FUNCTION_BLOCK FB_CH_List EXTENDS FB_CH_Object IMPLEMENTS I_CH_LIST, I_CH_List_Dublicate
VAR
	{attribute 'hide'}
	nObjectCount			: UDINT;
	{attribute 'hide'}
	nIdxNextObject			: UDINT;
	{attribute 'hide'}
	nIdxLastRestoreValues : ARRAY [0..(MAX_CTS_RESTORE_VALUES+1)] OF UDINT;
	{attribute 'hide'}
	nIdxRestore				: UDINT;
	{attribute 'hide'}
	aObjects				: ARRAY [1..BaseParameterlist.MAX_OBJECTS] OF I_CH_Object;
END_VAR
VAR CONSTANT
	{attribute 'hide'}
	MAX_CTS_RESTORE_VALUES : UINT := 20;
END_VAR

//Add all objects from the list in to this list
METHOD PUBLIC AddList : HRESULT
VAR_INPUT
	ipList	: I_CH_List;
END_VAR
VAR
	hr : HRESULT;
	ipListDublicate : I_CH_List_Dublicate;
	refRemoteList : REFERENCE TO ARRAY [1..BaseParameterlist.MAX_OBJECTS] OF I_CH_Object;
	pRemoteList : PVOID;
END_VAR
VAR_INST
	{attribute 'hide'}
	fbAlarmInvalideInputparm : FB_TcAlarm;
	{attribute 'hide'}
	fbAlarmListToSmall : FB_TcAlarm;
END_VAR
// Invalide input
IF ipList = 0 THEN
	fbAlarmInvalideInputparm.CreateEx(stEventEntry:= TC_EVENTS.CHALET_Base_Events.Invalide_Inputparameter, 
							ipSourceInfo := THIS^.fbSourceInfo, 
							bWithConfirmation := FALSE);
	fbAlarmInvalideInputparm.ipArguments.Clear().AddStringByValue('ipList');
	fbAlarmInvalideInputparm.Raise(0);	

	AddList := S_FALSE;
	RETURN;
END_IF


// This list is to small
IF (ipList.Size + THIS^.Size) > BaseParameterlist.MAX_OBJECTS THEN
	fbAlarmListToSmall.CreateEx(stEventEntry:= TC_EVENTS.CHALET_Base_Events.ListIsToSmall, 
							ipSourceInfo := THIS^.fbSourceInfo, 
							bWithConfirmation := FALSE);
	fbAlarmListToSmall.Raise(0);	

	AddList := S_FALSE;
	RETURN;
END_IF


//Done nothing to add
IF ipList.Size = 0 THEN
	AddList := S_OK;
	RETURN;
END_IF


//Check if the list has an optional I_CH_List_Dublicate interface. If so use the faste memcpy, else use default list commands
IF __QUERYINTERFACE(ipList, ipListDublicate) AND_THEN __ISVALIDREF(ipListDublicate.Content) THEN
	refRemoteList REF= ipListDublicate.Content;
	pRemoteList := ADR(refRemoteList);
	Tc2_System.MEMCPY(destAddr:= ADR(THIS^.aObjects[(THIS^.nObjectCount+1)]), srcAddr:= pRemoteList, n:= (SIZEOF(THIS^.aObjects[1])*ipList.Size) );
	THIS^.nObjectCount := ipList.Size + THIS^.nObjectCount; //Set size of List
ELSE
	ipList.ResetIterator();
	WHILE ipList.HasNextObject() DO
		hr := THIS^.AddObject(ipList.GetNextObject());
		IF hr <> S_OK THEN
			//Error
			AddList := hr;
			RETURN;
		END_IF
	END_WHILE
	ipList.RestoreIterator();
END_IF
END_METHOD

METHOD PUBLIC AddObject : HRESULT
VAR_INPUT
	iChObject	: I_CH_Object;
END_VAR
VAR_INST
	{attribute 'hide'}
	fbAlarmListFull : FB_TcAlarm;
END_VAR
IF iChObject = 0 THEN
	AddObject := S_FALSE;
	RETURN;
END_IF


//Error if list is allready full
IF nObjectCount >= BaseParameterlist.MAX_OBJECTS THEN
	fbAlarmListFull.CreateEx(stEventEntry:= TC_EVENTS.CHALET_Base_Events.ListIsFull, 
							ipSourceInfo := THIS^.fbSourceInfo, 
							bWithConfirmation := FALSE);
	fbAlarmListFull.ipArguments.Clear().AddStringByValue(iChObject.LUID);
	fbAlarmListFull.Raise(0);
	AddObject := S_FALSE;
	RETURN;
END_IF


//Add to list
nObjectCount := nObjectCount + 1;
aObjects[nObjectCount] := iChObject;

AddObject := S_OK;
END_METHOD

METHOD PUBLIC Clear : BOOL
VAR
	nIdx : UDINT;
END_VAR
Tc2_System.MEMSET(	destAddr	:= ADR(aObjects[1]), 
					fillByte	:= 0, 
					n			:= SIZEOF(aObjects[1])*BaseParameterlist.MAX_OBJECTS);


nObjectCount	:= 0;
nIdxNextObject	:= 0;
END_METHOD

//DEBUG only. View content for easy debug. Do not use this property
{attribute 'monitoring':='call'}
PROPERTY Content : REFERENCE TO ARRAY [1..BaseParameterlist.MAX_OBJECTS] OF I_CH_Object
GET
Content REF= THIS^.aObjects;
END_GET
END_PROPERTY

METHOD Duplicate : BOOL
VAR_INPUT
	ipListCopyFrom : I_CH_LIST;
END_VAR
VAR
	ipThisList : I_CH_LIST := THIS^;
	hr : HRESULT;
	ipListDublicate : I_CH_List_Dublicate;
	refRemoteList : REFERENCE TO ARRAY [1..BaseParameterlist.MAX_OBJECTS] OF I_CH_Object;
	pRemoteList : PVOID;
END_VAR
VAR_INST
	{attribute 'hide'}
	fbAlarmInvalideInputparm : FB_TcAlarm;
	{attribute 'hide'}
	fbAlarmListToSmall : FB_TcAlarm;
END_VAR
//New list equals this list
IF ipListCopyFrom = ipThisList THEN
	//Do Nothing - Successfull
	Duplicate := TRUE;
	RETURN;
END_IF

THIS^.Clear();

// Invalide input
IF ipListCopyFrom = 0 THEN
	fbAlarmInvalideInputparm.CreateEx(stEventEntry:= TC_EVENTS.CHALET_Base_Events.Invalide_Inputparameter, 
							ipSourceInfo := THIS^.fbSourceInfo, 
							bWithConfirmation := FALSE);
	fbAlarmInvalideInputparm.ipArguments.Clear().AddStringByValue('ipListCopyFrom');
	fbAlarmInvalideInputparm.Raise(0);	

	Duplicate := FALSE;
	RETURN;
END_IF


// This list is to small
IF ipListCopyFrom.Size > BaseParameterlist.MAX_OBJECTS THEN
	fbAlarmListToSmall.CreateEx(stEventEntry:= TC_EVENTS.CHALET_Base_Events.ListIsToSmall, 
							ipSourceInfo := THIS^.fbSourceInfo, 
							bWithConfirmation := FALSE);
	fbAlarmListToSmall.Raise(0);	
	Duplicate := FALSE;
	RETURN;
END_IF


//Done nothing to add
IF ipListCopyFrom.Size = 0 THEN
	Duplicate := TRUE;
	RETURN;
END_IF


//Check if the list has an optional I_CH_List_Dublicate interface. If so use the faste memcpy, else use list commands
IF __QUERYINTERFACE(ipListCopyFrom, ipListDublicate) AND_THEN __ISVALIDREF(ipListDublicate.Content) THEN
	refRemoteList REF= ipListDublicate.Content;
	pRemoteList := ADR(refRemoteList);
	Tc2_System.MEMCPY(destAddr:= ADR(THIS^.aObjects), srcAddr:= pRemoteList, n:= (SIZEOF(THIS^.aObjects[1])*ipListCopyFrom.Size) );
	THIS^.nObjectCount := ipListCopyFrom.Size; //Set size of List
ELSE
	ipListCopyFrom.ResetIterator();
	WHILE ipListCopyFrom.HasNextObject() DO
		hr := THIS^.AddObject(ipListCopyFrom.GetNextObject());
		IF hr <> S_OK THEN
			//Error
			Duplicate := FALSE;
			RETURN;
		END_IF
	END_WHILE
	ipListCopyFrom.RestoreIterator();	
END_IF


Duplicate := TRUE;
END_METHOD

METHOD PUBLIC FindLUID : I_CH_OBJECT
VAR_INPUT
	sLUID	: STRING;
END_VAR
VAR
	nIdx : UDINT;
END_VAR
FOR nIdx := 1 TO nObjectCount DO
	IF aObjects[nIdx] <> 0 AND_THEN aObjects[nIdx].LUID = sLUID THEN
		FindLUID := aObjects[nIdx];
		EXIT;
	END_IF
END_FOR
END_METHOD

METHOD FindOID : I_CH_OBJECT
VAR_INPUT
	nOID	: OTCID;
END_VAR
VAR
	nIdx : UDINT;
END_VAR
FOR nIdx := 1 TO nObjectCount DO
	IF aObjects[nIdx] <> 0 AND_THEN aObjects[nIdx].OID = nOID THEN
		FindOID := aObjects[nIdx];
		EXIT;
	END_IF
END_FOR
END_METHOD

METHOD FindOIDString : I_CH_OBJECT
VAR_INPUT
	sOID	: STRING;
END_VAR
VAR
	nIdx : UDINT;
END_VAR
FOR nIdx := 1 TO nObjectCount DO
	IF aObjects[nIdx] <> 0 AND_THEN DWORD_TO_HEXSTR(TO_DWORD(aObjects[nIdx].OID),0,FALSE) = sOID THEN
		FindOIDString := aObjects[nIdx];
		EXIT;
	END_IF
END_FOR
END_METHOD

METHOD PUBLIC GetNextObject : I_CH_Object
VAR_INPUT
END_VAR
VAR_INST
	{attribute 'hide'}
	fbAlarmInvalideEndOfList : FB_TcAlarm;
END_VAR
nIdxNextObject := nIdxNextObject + 1;


IF nIdxNextObject > nObjectCount THEN
	//Error!
	fbAlarmInvalideEndOfList.CreateEx(stEventEntry:= TC_EVENTS.CHALET_Base_Events.Invalive_EndOfList, 
							ipSourceInfo := THIS^.fbSourceInfo, 
							bWithConfirmation := FALSE);
	fbAlarmInvalideEndOfList.ipArguments.Clear().AddStringByValue('.GetNextObject()');
	fbAlarmInvalideEndOfList.Raise(0);
	RETURN;
END_IF




GetNextObject := aObjects[nIdxNextObject];
END_METHOD

METHOD GetObjectWithHighestNumber : I_CH_Object

VAR
	nIdx : UDINT;
	nMaxSortNbr : UDINT;
END_VAR




//Check array until a match
FOR nIdx := 1 TO THIS^.nObjectCount DO
	IF THIS^.aObjects[nIdx].SortOrderInList >= nMaxSortNbr THEN
		GetObjectWithHighestNumber := THIS^.aObjects[nIdx];
		nMaxSortNbr := THIS^.aObjects[nIdx].SortOrderInList;
	END_IF
END_FOR
END_METHOD

METHOD GetObjectWithLowestNumber : I_CH_Object
VAR
	nIdx : UDINT;
	nMinSortNbr : UDINT := GVL_Datatypes.cMaxUDint;
END_VAR
//Check array until a match
FOR nIdx := 1 TO THIS^.nObjectCount DO
	IF THIS^.aObjects[nIdx].SortOrderInList <= nMinSortNbr THEN
		GetObjectWithLowestNumber := THIS^.aObjects[nIdx];
		nMinSortNbr := THIS^.aObjects[nIdx].SortOrderInList;
	END_IF
END_FOR
END_METHOD

METHOD GetRandomObject : I_CH_Object
VAR_INPUT
END_VAR

VAR_INST
	{attribute 'hide'}
	fbDRAN : DRAND;
END_VAR

VAR
	nRandomIdx : UDINT;
END_VAR
//Check if not Empty
IF UDINT_TO_BOOL(nObjectCount) THEN
	// Generate number 0..1
	fbDRAN(Seed:= 42);
	
	// 1..Size   = ((0..1)*(Size-1))+1
	nRandomIdx := LREAL_TO_UDINT(fbDRAN.Num * (nObjectCount-1))+1;
	
	GetRandomObject := aObjects[nRandomIdx];
	
END_IF
END_METHOD

METHOD PUBLIC HasNextObject : BOOL
VAR_INPUT
END_VAR
HasNextObject := (nIdxNextObject < nObjectCount) AND_THEN (aObjects[nIdxNextObject+1] <> 0);
END_METHOD

METHOD Initialize : HRESULT //This method calls the respective Initialize method of all contained objects
VAR_INPUT
END_VAR
VAR
	hr : HRESULT;
	nIdx : UDINT;
END_VAR
//FOR each element
FOR nIdx := 1 TO nObjectCount DO
	// DO Init
	hr := GetMostSignificant(hr, aObjects[nIdx].Initialize());
END_FOR


Initialize := hr;
END_METHOD

{attribute 'monitoring':='call'}
PROPERTY PUBLIC IsEmpty : BOOL
GET
IsEmpty := (nObjectCount = 0);
END_GET
END_PROPERTY

{attribute 'monitoring':='call'}
PROPERTY PUBLIC IsFull : BOOL
GET
IsFull := (nObjectCount = BaseParameterlist.MAX_OBJECTS);
END_GET
END_PROPERTY

METHOD PUBLIC LUIDInList : BOOL
VAR_INPUT
	sLUID	: STRING;
END_VAR
VAR
	nIdx : UDINT;
END_VAR
//Check array until a match
FOR nIdx := 1 TO THIS^.nObjectCount DO
	IF THIS^.aObjects[nIdx].LUID = sLUID THEN
		LUIDInList := TRUE;
		EXIT;
	END_IF
END_FOR
END_METHOD

METHOD PUBLIC ObjectInList : BOOL
VAR_INPUT
	iChObject	: I_CH_Object;
END_VAR
VAR
	nIdx : UDINT;
END_VAR
//Check array until a match
FOR nIdx := 1 TO THIS^.nObjectCount DO
	IF THIS^.aObjects[nIdx] = iChObject THEN
		ObjectInList := TRUE;
		EXIT;
	END_IF
END_FOR
END_METHOD

METHOD PUBLIC OIDInList : BOOL
VAR_INPUT
	nOID	: OTCID;
END_VAR
VAR
	nIdx : UDINT;
END_VAR
//Check array until a match
FOR nIdx := 1 TO THIS^.nObjectCount DO
	IF THIS^.aObjects[nIdx].OID = nOID THEN
		OIDInList := TRUE;
		EXIT;
	END_IF
END_FOR
END_METHOD

METHOD RemoveAllDuplicateObjects : HRESULT
VAR_INPUT
END_VAR
VAR
	nIdx : UDINT;
	fbTempList : FB_CH_List;
	fbFoundDublicateObjects : FB_CH_List;
END_VAR
//Check eacht element in array, if allready was added in temp list. if found, delete
FOR nIdx := 1 TO THIS^.nObjectCount DO
	
	//check if allready was found
	IF fbTempList.ObjectInList(THIS^.aObjects[nIdx]) THEN
		//Found, add to an list to delete in next step
		fbFoundDublicateObjects.AddObject(THIS^.aObjects[nIdx]);	
	ELSE
		//Not found, add to list
		fbTempList.AddObject(THIS^.aObjects[nIdx]);	
	END_IF
END_FOR


//Delete in this list
fbFoundDublicateObjects.ResetIterator();
WHILE fbFoundDublicateObjects.HasNextObject() DO
	THIS^.RemoveObject(fbFoundDublicateObjects.GetNextObject());
END_WHILE
END_METHOD

METHOD PUBLIC RemoveObject : BOOL
VAR_INPUT
	iChObject	: I_CH_Object;
END_VAR

VAR
	nIdx			: UDINT;
END_VAR
RemoveObject := FALSE;

IF iChObject = 0 THEN
	RETURN;
END_IF

IF NOT THIS^.ObjectInList(iChObject) THEN
	RETURN;
END_IF

FOR nIdx := 1 TO nObjectCount DO
	IF aObjects[nIdx] = iChObject THEN
		aObjects[nIdx] := NULL;	
		
		nObjectCount := nObjectCount - 1;
		
		// Fill up the empty slot
		MEMMOVE(ADR(aObjects[nIdx]), ADR(aObjects[nIdx + 1]), SIZEOF(aObjects[nIdx]) * (BaseParameterlist.MAX_OBJECTS - nIdx));
	
		// If pos in list is less than ListIterator, then reduce Iterator
		IF nIdx <= nIdxNextObject THEN
			nIdxNextObject := nIdxNextObject -1;
		END_IF
		
		//Finish
		RemoveObject := TRUE;
		EXIT;
			
	END_IF
END_FOR
END_METHOD

METHOD PUBLIC ResetIterator : BOOL
VAR_INPUT
END_VAR
//Store the last few index for later restore if required - Shift array +1 step
MEMMOVE(srcAddr 	:= ADR(nIdxLastRestoreValues[0]), 
		destAddr 	:= ADR(nIdxLastRestoreValues[1]), 
		n 			:= (SIZEOF(nIdxNextObject)*MAX_CTS_RESTORE_VALUES));

//Store the last few index for later restore if required - Store last value
nIdxLastRestoreValues[0] := nIdxNextObject;


nIdxNextObject := 0;
END_METHOD

//Restore the iterator to the value before the last reset. This is necessary if several while loops are placed inside each other
METHOD PUBLIC RestoreIterator : BOOL
VAR_INPUT
END_VAR
//Store the last few index for later restore if required - Restore
nIdxNextObject := nIdxLastRestoreValues[0];

//Store the last few index for later restore if required - Shift array -1 step
MEMMOVE(srcAddr 	:= ADR(nIdxLastRestoreValues[1]), 
		destAddr 	:= ADR(nIdxLastRestoreValues[0]), 
		n 			:= (SIZEOF(nIdxNextObject)*MAX_CTS_RESTORE_VALUES));
END_METHOD

{attribute 'monitoring':='call'}
PROPERTY PUBLIC Size : UDINT
GET
Size := nObjectCount;
END_GET
END_PROPERTY

//Tthe entire list sorted BY ascending number. (small numbers AT the beginning).
//The FB_CH_Object.SortOrderInList is used
METHOD Sort : HRESULT
VAR
	fbCopyOfList : FB_CH_List;
	ipObjToAdd : I_CH_Object;
END_VAR
//TODO: use a smarter algorithm with less computational effort




//Create a copy of this list
fbCopyOfList.Duplicate(THIS^);

//Clear this List
THIS^.Clear();

//Add the smalest number to this list
WHILE NOT fbCopyOfList.IsEmpty DO
	ipObjToAdd := fbCopyOfList.GetObjectWithLowestNumber();
	fbCopyOfList.RemoveObject(ipObjToAdd);
	THIS^.AddObject(ipObjToAdd);
END_WHILE
END_METHOD

METHOD Update : HRESULT //This method calls the respective update method of all contained objects
VAR
	hr : HRESULT;
	nIdx : UDINT;
END_VAR
//FOR each element
FOR nIdx := 1 TO nObjectCount DO
	// DO Update
	hr := GetMostSignificant(hr, aObjects[nIdx].Update());
END_FOR

Update := hr;
END_METHOD

END_FUNCTION_BLOCK

(* stored: Version 1.1.0.1, ProductVersion 3.1.4024.13
   POU FB_CH_List: Id {af82aebc-49fb-4481-993c-d70fe342fe7b}, SpecialFunc None
   Folder Debug: Id {259d65e2-6e1e-4033-8d69-5bc4dd4162dc}
   Folder ID: Id {a6143771-4de3-44c7-bc68-b4e2d35fd4bb}
   Folder Iterator: Id {7b049406-fe3d-42b5-89c1-7ebd8af337c7}
   Folder List: Id {efee0648-7eeb-4629-a7ed-ed0883e34030}
   Folder Object: Id {a7ed3d9e-a61a-4f2c-ab17-a49e9491f215}
   Folder Sort: Id {79aa9360-7172-439c-a273-476aab94443e}
   Method AddList: Id {d78f867b-e215-47dc-8272-5375fc11c8aa}
   Method AddObject: Id {ba744631-6ed0-4654-afee-3bfb932f232e}
   Method Clear: Id {73a02d65-2240-453e-a05b-659da650929d}
   Property Content: Id {17a20f40-c58c-42c2-aa35-66426f827655}
   Get Get: Id {d7a6b570-d748-455b-b378-9402673b3fb9}
   Method Duplicate: Id {36ff03d9-f7f5-49fd-857d-d99230d76119}
   Method FindLUID: Id {bc53e504-4d0c-4529-99d5-eee1f228239e}
   Method FindOID: Id {dcfd7f35-5592-4006-a139-3f9b322e26fc}
   Method FindOIDString: Id {bd44922b-450f-4b2f-bff7-d80428deade7}
   Method GetNextObject: Id {9ac6a4ec-048a-41e7-8a25-6c35c5ccb4d9}
   Method GetObjectWithHighestNumber: Id {ee81c51d-e2a2-43f0-9d42-10583248672c}
   Method GetObjectWithLowestNumber: Id {480d6024-da5c-4fb7-b6e9-7e94d73bd63d}
   Method GetRandomObject: Id {059b06dd-1f8b-4613-91de-50b7deb695fa}
   Method HasNextObject: Id {f8cb30ca-df34-4d67-85ef-f037614e067b}
   Method Initialize: Id {0433ca42-cba8-4876-af3c-f03841c3e69c}
   Property IsEmpty: Id {a58263fb-723e-4a96-8e1d-0843aa6cf381}
   Get Get: Id {47ab9808-3a1b-42c6-af29-c8e033e56da7}
   Property IsFull: Id {13a50413-ac00-484b-9332-500f70a60fe9}
   Get Get: Id {f560e3e3-ef8b-4ce8-b600-b0a9539508a0}
   Method LUIDInList: Id {89be4f5c-cb32-485e-87fc-ad951f5ab246}
   Method ObjectInList: Id {ecb05561-854b-4c37-ad37-3931b803da52}
   Method OIDInList: Id {1d43281c-110b-40c2-9c10-7cc6626d961e}
   Method RemoveAllDuplicateObjects: Id {fc8edc33-4d26-4376-ab23-b949c4c5d07f}
   Method RemoveObject: Id {2fbae86e-dd36-4e65-be68-63238054e89a}
   Method ResetIterator: Id {cf281138-b754-4d58-b0fb-8bfa602e34ce}
   Method RestoreIterator: Id {c0e73554-72a9-4fcf-ac42-2c657f276289}
   Property Size: Id {525ee8bc-7c1a-4cc4-9f59-cbf67c4a00b1}
   Get Get: Id {4583acbd-69b9-4373-8a95-f8bfb667dce5}
   Method Sort: Id {c9a98106-02cf-4336-9ba6-b62d16a29420}
   Method Update: Id {d0b62ac1-d7ee-4878-a622-e34d7fd6ea2d} *)
